// TODO rename + your HAL signals (outputs + feedback sensors), Core §3.6
TYPE ST_TemplateHal :
STRUCT
    OutA : BOOL;
    FbA  : BOOL;
END_STRUCT
END_TYPE

(* stored: Version 1.1.0.1, ProductVersion 3.1.4024.12
   DUT ST_TemplateHal: Id {346f01d0-b85d-4e94-bb99-4129b4f72d3d} *)
